PROGRAM MAIN
VAR
END_VAR

END_PROGRAM

(* stored: Version 1.1.0.1
   POU MAIN: Id {1c8bd6f4-6c72-4c53-9ec1-6e915895e7a9} *)
